# EPICS alarm handler configuration: alh_files/mgnt_bsyA_ycor.alhConfig
GROUP NULL YCOR:BSYA:MG01
   $COMMAND edm -x -eolc -noedit mgnt_bsy0_ycor.edl
$ALIAS YCOR
$GUIDANCE
BSY0 YCOR
   Group Name: YCOR:BSYA:MG01
   Summary PV:  YCOR:BSYA:MG01:STATSUMY
$END

GROUP YCOR:BSYA:MG01  YCOR:BSYA:333
   $COMMAND edm -x -eolc -noedit -m "DEV=YCOR:BSYA:333,PDEV=PS:BSY0:7,IOC=YCOR:BSYA:333" mgnt_unit2.edl
CHANNEL    YCOR:BSYA:333    YCOR:BSYA:333:STATMSG   -----
   $FORCEPV YCOR:BSYA:333:STATMSGSV -DATL 1 0
